VAR_GLOBAL
////////////////////////////////////////:	///////////////////////////////////////////////////
/////////////////////////////////////////////////////////////////////////////////////GENERIC/////////////////////////////////////////////////////////////////////////////////////

	// PowerUP 
	tonSystemPowerUP				:TON;
	tSystemPowerUP_Time				:TIME								:=T#3S;
	bSystemPoweringUP				:BOOL								:=TRUE; //Global System PowerUP Flag
	
	fbSystemShutDown     	        : NT_Shutdown;
	stButtonsLamps					: ST_ButtonsLamps;
	rtrigButton             		: ARRAY[1..3] OF Tc2_Standard.R_TRIG;
	ftrigButton             		: ARRAY[1..3] OF Tc2_Standard.F_TRIG; 
	stPuls							: ST_Puls;		

	stCycleDataNest1				: ST_CycleData;
	stCycleDataNest2				: ST_CycleData;
	
	bWriteNest1						: BOOL;
	bWriteNest2						: BOOL;
	bCSVDone						: BOOL;
	bCSVReady						: BOOL;
	bAutocycleIDLE					: BOOL;
	bDoorOpenedFlag					: BOOL;
	
	bRejectPartFault				: BOOL;
	
	bCSVError						: BOOL;
	
	NetAmsIdLocal        	       	: T_AmsNetId;
	bReadAMSNetID					: BOOL;
	fbGetLocalAMSNetID				: FB_GetLocalAmsNetId;
	
	fbGetDeviceNetId				: IOF_GetDeviceNetId;
	NetAmsIdDevice					: T_AmsNetId;
	
	bOpenDoorCycleFault				: BOOL;
	bProcessDoorClosed				: BOOL;
	
	bPartPresentNest1				: BOOL;
	bPartPresentNest2				: BOOL;
	
	stTester						: ST_Tester;

	
/////////////////////////////////////////////////////////////////////////////////////Event Log/////////////////////////////////////////////////////////////////////////////////////
	
	stStationEvents				: ARRAY[0..4] OF  ST_StationEvents;//0: GENERAL
																	//1: Leak Test
																	//2: Height Test
																	//3: Vision 
																	//4: Cylinders
																	
																	
	astActiveEvents				: ARRAY [0..50] OF ST_ActiveEvents;
	stEventsAssigment			: ST_EventsAssigmentGeneral;
	bMachineMessages			: BOOL;
	sMachineMessage				: STRING;

/////////////////////////////////////////////////////////////////////////////////////MACHINE CONTROL////////////////////////////////////////////////////////////////////////////
	
	stMachineStatus					: ST_MachineStatus;	
	stMasterCtrl					: ST_MasterCTRL;
	bStatisticsTest					: ARRAY[0..5] OF  BOOL;
	
	
////////////////////////////////////////////////////////////////////////////////////SYSTEM////////////////////////////////////////////////////////////////////////////

	stSystemTime				: TIMESTRUCT;
	sSystemTime					: STRING(255);
	sSystemDate					: STRING(255);

////////////////////////////////////////////////////////////////////////////////////SAFETY////////////////////////////////////////////////////////////////////////////

	bDoorClosingFlag				: BOOL;
	bDoorClosingInitFlag			: BOOL;
	bDoorOpeningFlag				: BOOL;
	bProcessDoorClosedConditionFlag	: BOOL;
	tonSafety						: TON;
	bProcessCylinderSafetyPosition	: BOOL;
	bProcessDoorUpInitialising		: BOOL;
	
END_VAR

(* stored: Version 1.1.0.1, ProductVersion 3.1.4026.18
   GVL GVL_Master: Id {ff1c03dd-d56c-490f-bced-572c30dff423} *)
